// TIA Portal V20 export
// export: Created 2026-04-11T06:02:30.2090393Z, ExportSetting WithDefaults, DisplayName Totally Integrated Automation Portal, DisplayVersion V20, DisplayName TIA Portal Openness, DisplayVersion V20, DisplayName TIA Portal Version Control Interface, DisplayVersion V20, DisplayName STEP 7 Professional, DisplayVersion V20, DisplayName STEP 7 Safety, DisplayVersion V20, DisplayName WinCC Basic/Comfort/Advanced, DisplayVersion V20, DisplayName WinCC Unified, DisplayVersion V20
TYPE "udtHMI_SiwarexControl"
// stored: IsFailsafeCompliant false
   STRUCT
      iMode : Int;   // Current mode
      iErrorCode { ExternalWritable := 'False'} : Int;   // Error code
      iStatus { ExternalWritable := 'False'} : Int;   // Status for HMI display
      iModuleAddress { S7_SetPoint := 'True'} : Int;   // IO start address of the module
      bPB_TareLoadCell : Bool;   // PB to tare the load cell
      bPBEN_TareLoadCell { ExternalWritable := 'False'} : Bool;   // Enable taring of the load cell
      bPB_DeleteTareValue : Bool;   // PB to delete current tare
      bPB_ResetError : Bool;   // PB to reset error
      bError { ExternalWritable := 'False'} : Bool;   // Error exists
      rActualWeight { ExternalWritable := 'False'} : Real;   // Current weight measured by load cell
      rManualWeight { S7_SetPoint := 'True'} : Real;   // Manual override weight from HMI
   END_STRUCT;
END_TYPE
